PROGRAM P_RunClock
VAR
	
	fbClock : FB_Clock;
	
END_VAR


fbClock(
	bStartEnable := G_HMI.bstepp_button,
	fTimeStep := G_Parameters.fTimeStep,
	
	fTime => G_OPC.fTime
);

END_PROGRAM

(* stored: Version 1.1.0.1
   POU P_RunClock: Id {3607f292-5366-4b7c-810f-569374c051f5}, SpecialFunc None *)
